PROGRAM MAIN
VAR
	fbCar 	: FB_Beckhoff_EV;
END_VAR

fbCar();

END_PROGRAM

(* stored: Version 1.1.0.1, ProductVersion 3.1.4024.4
   POU MAIN: Id {727f5f4a-fdfc-4f92-bb10-1d13c50fce2b}, SpecialFunc None *)
